{attribute 'qualified_only'}
VAR_GLOBAL
eStatus : E_Status;
stVisuParam : ST_VisuParam;
eMode : E_Mode;
END_VAR

(* stored: Version 1.1.0.1, ProductVersion 3.1.4024.12
   GVL HMI: Id {2c17b807-7a1f-4985-aea0-7bd489cec1d7} *)
